PROGRAM MAIN
VAR
    // Carro: FB_Carro_DRC_LD;
    Carro: FB_Carro_GRF_SFC;
    // Carro: FB_Carro_GRF_ST;
    // Carro: FB_Carro_GRF_LD;
END_VAR

Carro();

END_PROGRAM

(* stored: Version 1.1.0.1, ProductVersion 3.1.4024.16
   POU MAIN: Id {7c37925b-362c-4ebf-880c-ca7e46ea3b81}, SpecialFunc None *)
